// TIA Portal V19 export
TYPE "LAF_typeEmCommands"
// Commands for the equipment module
// stored: Access Published
   STRUCT
      enable : Bool;   // Enable the equipment module
      acknowledge : Bool;   // Acknowledge the equipment module
      disableAlarms : Bool;   // Disable the alarms of the equipment module
      activateSimulation : Bool;   // Activate the simulation of the equipment module
      home : Bool;   // Home the equipment module
      moveToInitialPosition : Bool;   // Move the equipment module to initial position
      directModeControl : "LUC_typeModes";   // Direct Control of the Mode, if the equipment module is unlinked
      directStateControl : "LUC_typeStates";   // Direct Control of the State, if the equipment module is unlinked
   END_STRUCT;
END_TYPE
